% RSLogix 500 project Analog Pump Control with Alarms and Notifications.RSS, saved by version 8.30.00.16 %
PROJECT "UNTITLED"    % processor: Bul.1763 MicroLogix 1100 Series B %

PROGRAM FILES
  LAD 2 "MAIN"  4 rungs
  LAD 3 "IO"  4 rungs
  LAD 4 "CONTROLS"  7 rungs
  LAD 5 "ALARMS"  7 rungs

DATA FILES
  O0 OUTPUT  5 elements
  I1 INPUT  14 elements
  S2 STATUS  66 elements
  B3 BINARY  1 elements
  T4 TIMER  4 elements
  C5 COUNTER  1 elements
  R6 CONTROL  1 elements
  N7 INTEGER  1 elements
  F8 FLOAT  1 elements

LADDER 2 "MAIN"
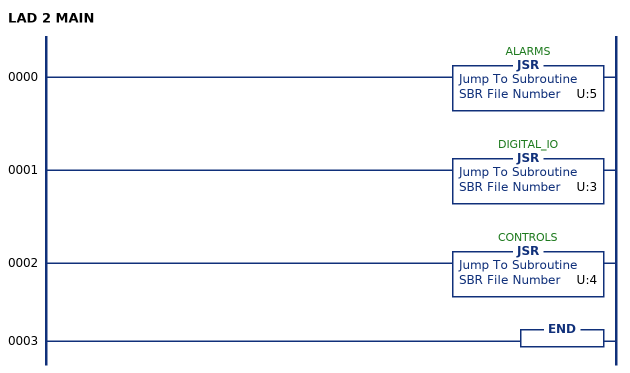
% Rung: 0 %
SOR JSR U:5 EOR
%   U:5  "ALARMS" %
% Rung: 1 %
SOR JSR U:3 EOR
%   U:3  "DIGITAL_IO" %
% Rung: 2 %
SOR JSR U:4 EOR
%   U:4  "CONTROLS" %
% Rung: 3 %
SOR END EOR

LADDER 3 "IO"
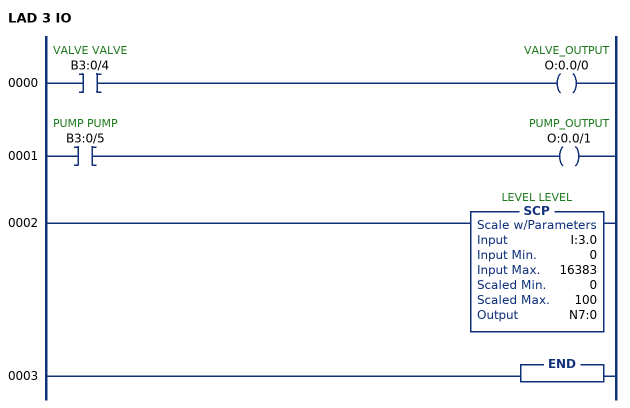
% Rung: 0 %
SOR XIC B3:0/4 OTE O:0.0/0 EOR
%   B3:0/4  VALVE  "VALVE" %
%   O:0.0/0  "VALVE_OUTPUT" %
% Rung: 1 %
SOR XIC B3:0/5 OTE O:0.0/1 EOR
%   B3:0/5  PUMP  "PUMP" %
%   O:0.0/1  "PUMP_OUTPUT" %
% Rung: 2 %
SOR SCP I:3.0 0 16383 0 100 N7:0 EOR
%   I:3.0  "LEVEL_SENSOR_INPUT" %
%   N7:0  LEVEL  "LEVEL" %
% Rung: 3 %
SOR END EOR

LADDER 4 "CONTROLS"
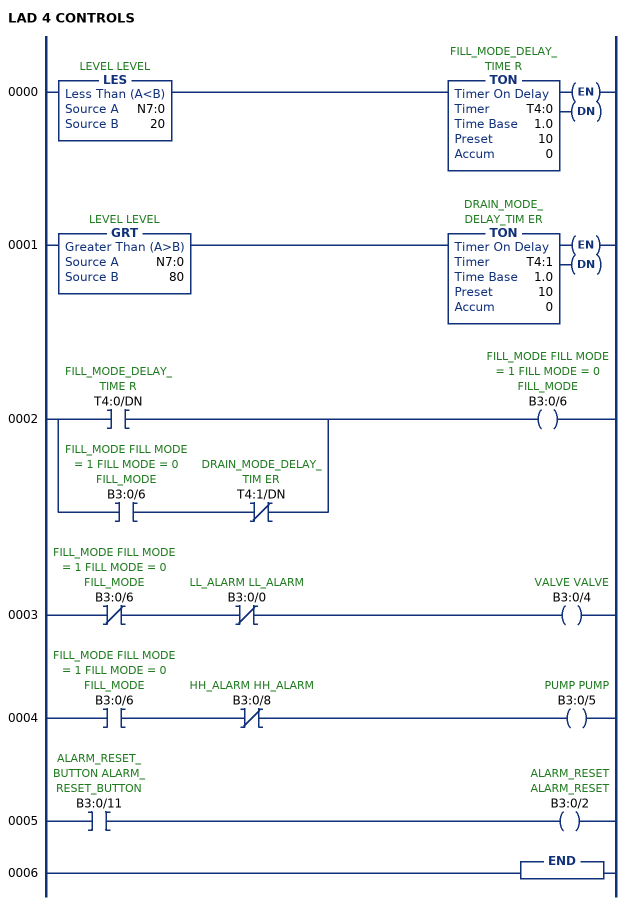
% Rung: 0 %
SOR LES N7:0 20 TON T4:0 1.0 10 0 EOR
%   N7:0  LEVEL  "LEVEL" %
%   T4:0  "FILL_MODE_DELAY_TIME R" %
% Rung: 1 %
SOR GRT N7:0 80 TON T4:1 1.0 10 0 EOR
%   N7:0  LEVEL  "LEVEL" %
%   T4:1  "DRAIN_MODE_DELAY_TIM ER" %
% Rung: 2 %
SOR BST XIC T4:0/DN NXB XIC B3:0/6 XIO T4:1/DN BND OTE B3:0/6 EOR
%   T4:0  "FILL_MODE_DELAY_TIME R" %
%   B3:0/6  FILL_MODE  "FILL_MODE FILL MODE = 1 FILL MODE = 0" %
%   T4:1  "DRAIN_MODE_DELAY_TIM ER" %
% Rung: 3 %
SOR XIO B3:0/6 XIO B3:0/0 OTE B3:0/4 EOR
%   B3:0/6  FILL_MODE  "FILL_MODE FILL MODE = 1 FILL MODE = 0" %
%   B3:0/0  LL_ALARM  "LL_ALARM" %
%   B3:0/4  VALVE  "VALVE" %
% Rung: 4 %
SOR XIC B3:0/6 XIO B3:0/8 OTE B3:0/5 EOR
%   B3:0/6  FILL_MODE  "FILL_MODE FILL MODE = 1 FILL MODE = 0" %
%   B3:0/8  HH_ALARM  "HH_ALARM" %
%   B3:0/5  PUMP  "PUMP" %
% Rung: 5 %
SOR XIC B3:0/11 OTE B3:0/2 EOR
%   B3:0/11  ALARM_RESET_BUTTON  "ALARM_RESET_BUTTON" %
%   B3:0/2  ALARM_RESET  "ALARM_RESET" %
% Rung: 6 %
SOR END EOR

LADDER 5 "ALARMS"
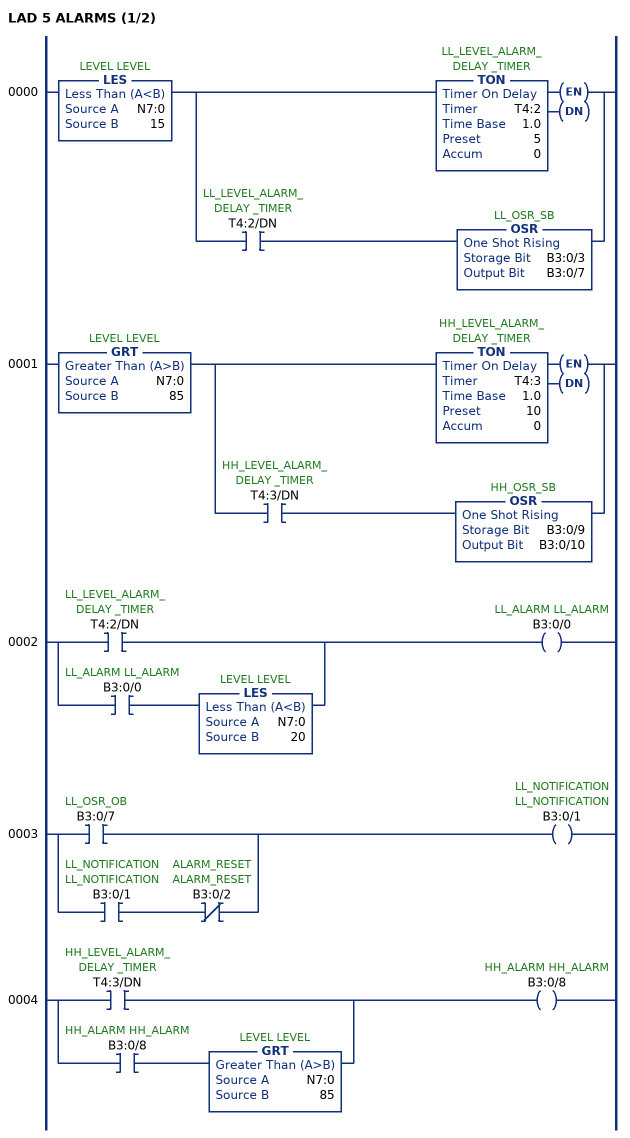
% Rung: 0 %
SOR LES N7:0 15 BST TON T4:2 1.0 5 0 NXB XIC T4:2/DN OSR B3:0/3 B3:0/7 BND EOR
%   N7:0  LEVEL  "LEVEL" %
%   T4:2  "LL_LEVEL_ALARM_DELAY _TIMER" %
%   B3:0/3  "LL_OSR_SB" %
%   B3:0/7  "LL_OSR_OB" %
% Rung: 1 %
SOR GRT N7:0 85 BST TON T4:3 1.0 10 0 NXB XIC T4:3/DN OSR B3:0/9 B3:0/10 BND EOR
%   N7:0  LEVEL  "LEVEL" %
%   T4:3  "HH_LEVEL_ALARM_DELAY _TIMER" %
%   B3:0/9  "HH_OSR_SB" %
%   B3:0/10  "HH_ALARM_OB" %
% Rung: 2 %
SOR BST XIC T4:2/DN NXB XIC B3:0/0 LES N7:0 20 BND OTE B3:0/0 EOR
%   T4:2  "LL_LEVEL_ALARM_DELAY _TIMER" %
%   B3:0/0  LL_ALARM  "LL_ALARM" %
%   N7:0  LEVEL  "LEVEL" %
% Rung: 3 %
SOR BST XIC B3:0/7 NXB XIC B3:0/1 XIO B3:0/2 BND OTE B3:0/1 EOR
%   B3:0/7  "LL_OSR_OB" %
%   B3:0/1  LL_NOTIFICATION  "LL_NOTIFICATION" %
%   B3:0/2  ALARM_RESET  "ALARM_RESET" %
% Rung: 4 %
SOR BST XIC T4:3/DN NXB XIC B3:0/8 GRT N7:0 85 BND OTE B3:0/8 EOR
%   T4:3  "HH_LEVEL_ALARM_DELAY _TIMER" %
%   B3:0/8  HH_ALARM  "HH_ALARM" %
%   N7:0  LEVEL  "LEVEL" %

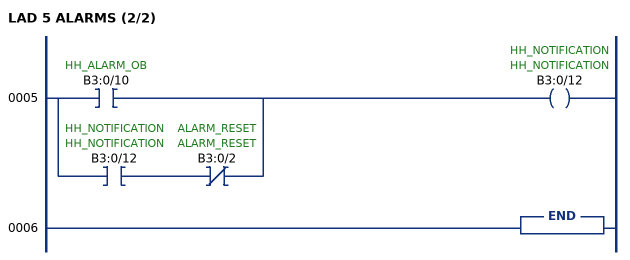
% Rung: 5 %
SOR BST XIC B3:0/10 NXB XIC B3:0/12 XIO B3:0/2 BND OTE B3:0/12 EOR
%   B3:0/10  "HH_ALARM_OB" %
%   B3:0/12  HH_NOTIFICATION  "HH_NOTIFICATION" %
%   B3:0/2  ALARM_RESET  "ALARM_RESET" %
% Rung: 6 %
SOR END EOR

OTHER DOCUMENTED ADDRESSES
  I:0  "LEVEL_SENSOR_INPUT"
  I:1.0/0  "LL_SWITCH_INPUT"
  I:1.0/1  "L_SWITCH_INPUT"
  I:1.0/2  "H_SWITCH_INPUT"
  I:1.0/3  "HH_SWITCH_INPUT"
  N7:0/0  "LEVEL"
  O:0  "VALVE_OUTPUT"

REVISION NOTES
  0: Added Alarm Reset Button

DATA TABLE (non-zero values as saved)
DATA T4
% .PRE .ACC %
% T4:0 % 10 0
% T4:1 % 10 0
% T4:2 % 5 0
% T4:3 % 10 0
DATA N7
% N7:0 % 90
